PROGRAM EM03_PalletOutfeed
VAR
END_VAR

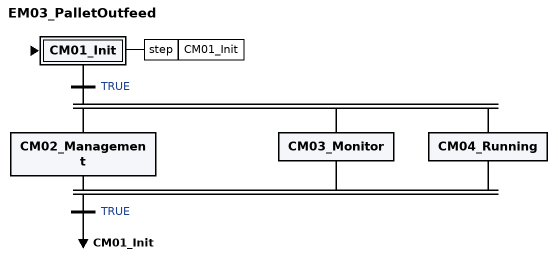
INITIAL_STEP CM01_Init:
    CM01_Init(N);  // step action
END_STEP
TRANSITION FROM CM01_Init TO (CM02_Management, CM03_Monitor, CM04_Running)
    := TRUE;
END_TRANSITION
STEP CM02_Management:
END_STEP
STEP CM03_Monitor:
END_STEP
STEP CM04_Running:
END_STEP
TRANSITION FROM (CM02_Management, CM03_Monitor, CM04_Running) TO CM01_Init
    := TRUE;
END_TRANSITION

ACTION CM01_Init:

END_ACTION

ACTION CM02_Management:
// NETWORK 1
END_ACTION

ACTION CM03_Monitor:
// NETWORK 1
END_ACTION

ACTION CM04_Running:
// NETWORK 1
END_ACTION

END_PROGRAM

(* stored: Version 1.1.0.1, ProductVersion 3.1.4024.9
   POU EM03_PalletOutfeed: Id {1ead50ca-4de4-4f6d-8438-948f52210416}, SpecialFunc None
   Action CM01_Init: Id {526f059e-73ed-4052-a587-ed837cbb56db}
   Action CM02_Management: Id {ccfd1d37-32ba-40fa-9af0-eb4610fdd98e}
   Action CM03_Monitor: Id {e72da1cd-be9e-4e54-ab5d-1c67755a1620}
   Action CM04_Running: Id {db79755e-476e-4f34-a009-28492eaf5ed4} *)
